ABB RobotStudio station: Project2.rsstnx

Station Project2 (saved by RobotStudio 23.2.10478.1)
Controller Steuerung1
  mechanical unit ROB_1: IRB1600_6_120__02, 6 joints, base frame (0, 0, 0) mm
Layout (positions relative to the parent item):
  - IRB1600_6_120__02 [mechanism, from %ABB.RobotStudio.Models.IRB1600%\IRB1600_6_120_G_02.rslib] at (0, 0, 0) mm; joint values [-1.249, 0.8715, -0.1121, 0, 0.8115, 1.8925] (rad or m)
  - Smart_Gripper_Servo_Fingers [mechanism, from %ABB.RobotStudio.Models.SmartGripper%\ABB_Smart_Gripper_Servo_Fingers.rslib] at (300, -900, 314.2) mm, rotated rx -180 ry 0 rz 0 deg; joint values [0] (rad or m)
  - Teil_1 [part], size 1000 x 500 x 50 mm
  - 1600_3str_h2 [part, from %ABB.RobotStudio.Models.Conveyors%\Conveyor 1600 3str h2.rslib] at (650, 0, 0) mm
  - Koordinatensystem_1 [frame] at (500, -500, 50) mm, rotated rx 0 ry 0 rz 180 deg
Attachment: Smart_Gripper_Servo_Fingers is attached to IRB1600_6_120__02 / Link6
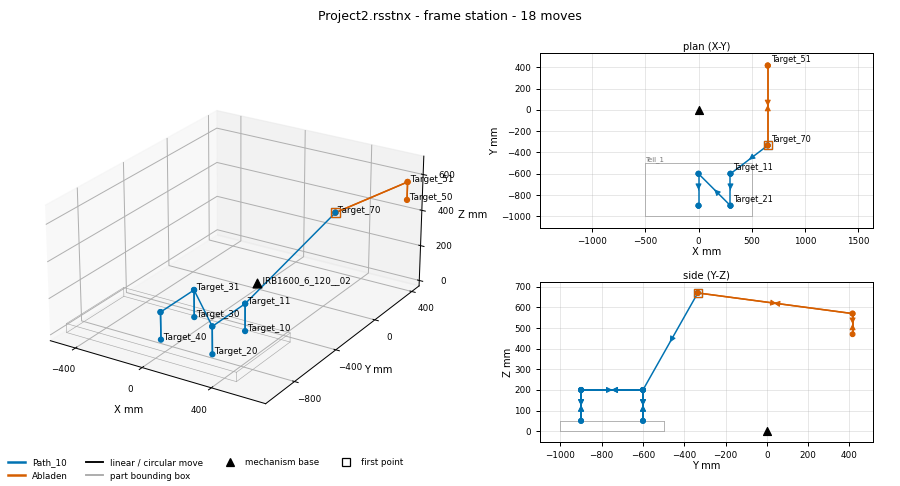
[picture p0: tool path of Project2.rsstnx in frame station, 18 of 18 moves have a stored position in this frame; points joined in program order, loops and branches not executed]
Targets, tools, work objects and paths stored in the station, written as RAPID:
! task T_ROB1
MODULE CalibData
  PERS tooldata Servo:=[TRUE,[[0,0,114.2],[1,0,0,0]],[0.215,[8.7,12.3,49.2],[1,0,0,0],0.00021,0.00024,0.00009]];
ENDMODULE

! task T_ROB1
MODULE Module1
  CONST robtarget Target_10:=[[300,-600,50],[0,1,0,0],[0,0,0,0],[9E+09,9E+09,9E+09,9E+09,9E+09,9E+09]];
  CONST robtarget Target_20:=[[300,-900,50],[0,1,0,0],[0,0,0,0],[9E+09,9E+09,9E+09,9E+09,9E+09,9E+09]];
  CONST robtarget Target_30:=[[0,-600,50],[0,1,0,0],[0,0,0,0],[9E+09,9E+09,9E+09,9E+09,9E+09,9E+09]];
  CONST robtarget Target_40:=[[0,-900,50],[0,1,0,0],[0,0,0,0],[9E+09,9E+09,9E+09,9E+09,9E+09,9E+09]];
  CONST robtarget Target_50:=[[650,415.688,470],[0,0,1,0],[0,0,0,0],[9E+09,9E+09,9E+09,9E+09,9E+09,9E+09]];
  CONST robtarget Target_60:=[[650,415.688,570],[0,0,1,0],[0,0,0,0],[9E+09,9E+09,9E+09,9E+09,9E+09,9E+09]];
  CONST robtarget Target_70:=[[650,-334.312,670],[0,0,1,0],[-1,0,-1,0],[9E+09,9E+09,9E+09,9E+09,9E+09,9E+09]];
  CONST robtarget Target_11:=[[300,-600,200],[0,1,0,0],[0,0,0,0],[9E+09,9E+09,9E+09,9E+09,9E+09,9E+09]];
  CONST robtarget Target_51:=[[650,415.688,570],[0,0,1,0],[0,0,0,0],[9E+09,9E+09,9E+09,9E+09,9E+09,9E+09]];
  CONST robtarget Target_31:=[[0,-600,200],[0,1,0,0],[0,0,0,0],[9E+09,9E+09,9E+09,9E+09,9E+09,9E+09]];
  CONST robtarget Target_41:=[[0,-900,200],[0,1,0,0],[0,0,0,0],[9E+09,9E+09,9E+09,9E+09,9E+09,9E+09]];
  CONST robtarget Target_21:=[[300,-900,200],[0,1,0,0],[0,0,0,0],[9E+09,9E+09,9E+09,9E+09,9E+09,9E+09]];
  PROC main()
    Path_10;
  ENDPROC
  PROC Path_10()
    MoveL Target_70,v1000,z100,Servo\WObj:=wobj0;
    MoveL Target_11,v1000,z100,Servo\WObj:=wobj0;
    MoveL Target_10,v100,fine,Servo\WObj:=wobj0;
    MoveL Target_11,v1000,z100,Servo\WObj:=wobj0;
    Abladen;
    MoveL Target_21,v1000,z100,Servo\WObj:=wobj0;
    MoveL Target_20,v100,fine,Servo\WObj:=wobj0;
    MoveL Target_21,v1000,z100,Servo\WObj:=wobj0;
    Abladen;
    MoveL Target_31,v1000,z100,Servo\WObj:=wobj0;
    MoveL Target_30,v100,fine,Servo\WObj:=wobj0;
    MoveL Target_31,v1000,z100,Servo\WObj:=wobj0;
    Abladen;
    MoveL Target_41,v1000,z100,Servo\WObj:=wobj0;
    MoveL Target_40,v100,fine,Servo\WObj:=wobj0;
    MoveL Target_41,v1000,z100,Servo\WObj:=wobj0;
    Abladen;
  ENDPROC
  PROC Abladen()
    MoveL Target_70,v1000,z100,Servo\WObj:=wobj0;
    MoveL Target_51,v1000,z100,Servo\WObj:=wobj0;
    MoveL Target_50,v100,fine,Servo\WObj:=wobj0;
    MoveL Target_51,v1000,z100,Servo\WObj:=wobj0;
    MoveL Target_70,v1000,z100,Servo\WObj:=wobj0;
  ENDPROC
ENDMODULE

